(* IEC 61131-3 sources: AXOpen/src/integrations/ctrl/src/Examples/AXOpen.AxoRemoteTask, 2 files *)

(* ---- AxoRemoteTaskDocuExample.st ---- *)
USING AXOpen.Core;

NAMESPACE AxoRemoteTaskDocuExamples
    //<IxRemoteTaskExample>
    CLASS MyRemoteTask EXTENDS AXOpen.Core.AxoRemoteTask
        VAR PUBLIC
            Message : STRING[254];
        END_VAR

        METHOD PUBLIC Invoke : IAxoTaskState
            VAR_INPUT
                LogMessage : STRING[254];
            END_VAR;
            Message := LogMessage;
            Invoke := SUPER.Invoke();
        END_METHOD

    END_CLASS
    //</IxRemoteTaskExample>
    CLASS RemoteTasks EXTENDS AXOpen.Core.AxoContext
        VAR PUBLIC
            _remoteTask : MyRemoteTask;
            _remoteTaskInvokeFromPlc : BOOL;
            _doneCounter : INT;
        END_VAR

        METHOD PROTECTED OVERRIDE Main

            //<IxTaskIntitialization>
            _remoteTask.Initialize(THIS); // THIS = IIContext
            //</IxTaskIntitialization>

            //<IxTaskInvoke>
            _remoteTask.Invoke('hello');
            //</IxTaskInvoke>

            //<IxTaskInvokeDone>
            IF(_remoteTask.Invoke('hello').IsDone()) THEN
                _doneCounter := _doneCounter + 1;
            END_IF;
            //</IxTaskInvokeDone>

            //<IxTaskInvokeDoneSeparatelly>

            // Fire & Forget
            _remoteTask.Invoke('hello');

            // What for done somwhere else
            IF(_remoteTask.IsDone()) THEN
                _doneCounter := _doneCounter + 1;
            END_IF;

            //</IxTaskInvokeDoneSeparatelly>

            //<IxTaskRunning>
            IF(_remoteTask.IsBusy()) THEN
                ;// Do something after task started
            END_IF;
            //</IxTaskRunning>

            //<IxTaskError>
            IF(_remoteTask.HasError()) THEN
                ;// Do something when an exception occurs on remote task.
            END_IF;
            //</IxTaskError>

            _remoteTask.Execute();

        END_METHOD
    END_CLASS
END_NAMESPACE

(* ---- AxoRemoteTaskExample.st ---- *)
USING AXOpen.Core;

NAMESPACE AxoRemoteTaskExamples

    CLASS MyRemoteTask EXTENDS AXOpen.Core.AxoRemoteTask
        VAR PUBLIC
            Message : STRING[254];
            Counter : INT;
        END_VAR

        METHOD PUBLIC Invoke : IAxoTaskState
            VAR_INPUT
                LogMessage : STRING[254];
                LogCounter : INT;
            END_VAR;
            Counter := LogCounter;
            Message := LogMessage;
            Invoke := SUPER.Invoke();
        END_METHOD

    END_CLASS

    CLASS RemoteTasks EXTENDS AxoContext
        VAR PUBLIC
            {#ix-set:AttributeName = "Click to execute this command"}
            _remoteTask : MyRemoteTask;
            {#ix-set:AttributeName = "Trigger from PLC"}
            _remoteTaskInvokeFromPlc : BOOL;
            _doneCounter : INT;
        END_VAR

        METHOD PROTECTED OVERRIDE Main
            _remoteTask.Initialize(THIS);

            IF(_remoteTaskInvokeFromPlc) THEN
                IF(_remoteTask.Invoke('hello', _doneCounter).IsDone()) THEN
                    _doneCounter := _doneCounter + 1;
                    _remoteTaskInvokeFromPlc := FALSE;
                END_IF;
            END_IF;
            _remoteTask.Execute();
        END_METHOD
    END_CLASS
END_NAMESPACE
